(*
	Get task cycle time in seconds.
*)
FUNCTION GetTaskCycleTime : LREAL
VAR_IN_OUT CONSTANT
	taskInfo: ARRAY[*] OF PlcTaskSystemInfo; // Just assign _TaskInfo as _TaskInfo cannot be accessed from lib :(
END_VAR

GetTaskCycleTime := UDINT_TO_LREAL(taskInfo[TC2_System.GETCURTASKINDEXEX()].CycleTime) / 10_000_000;

END_FUNCTION

(* stored: Version 1.1.0.1
   POU GetTaskCycleTime: Id {acded846-b650-4bf5-b83e-616dac5772c0}, SpecialFunc None *)
